(* IEC 61131-3 sources: io/test/Input, 8 files *)

(* ---- BinSignalExtTest.st ---- *)
USING AxUnit;
USING Simatic.Ax.IO.Input;
USING System.Timer;

NAMESPACE Simatic.Ax.IO.Input.Test

    /// Test fixture for BinSignalExt class
    /// Verifies extended binary signal functionality including:
    /// - All BinSignal features (signal reading, edge detection, inversion, quality status)
    /// - On-delay and off-delay timing functionality
    /// - Time-based signal filtering
    {TestFixture}
    CLASS BinSignalExtTest
        VAR
            o : BinSignalExt;  // Test object for BinSignalExt
            oStateLess : BinSignalExt;  // Stateless test object
        END_VAR

        /// Setup method called before each test
        /// Initializes test objects to ensure clean state
        {TestSetup}
        METHOD PUBLIC MyTestSetup
            o := oStateLess;
        END_METHOD

        /// Test basic signal reading - expects TRUE output when TRUE signal is read
        {Test}
        METHOD PUBLIC TestQ_And_expect_true
            o.ReadCyclic(signal := TRUE);
            Assert.Equal(expected := TRUE, actual := o.Q());
        END_METHOD

        {Test(isignal := FALSE, ienable := FALSE, idefault := FALSE, iexpq := FALSE, iexpqbad := TRUE)}
        {Test(isignal := FALSE, ienable := FALSE, idefault := TRUE, iexpq := TRUE, iexpqbad := TRUE)}
        {Test(isignal := FALSE, ienable := TRUE, idefault := FALSE, iexpq := FALSE, iexpqbad := FALSE)}
        {Test(isignal := FALSE, ienable := TRUE, idefault := TRUE, iexpq := FALSE, iexpqbad := FALSE)}

        {Test(isignal := TRUE, ienable := FALSE, idefault := FALSE, iexpq := FALSE, iexpqbad := TRUE)}
        {Test(isignal := TRUE, ienable := FALSE, idefault := TRUE, iexpq := TRUE, iexpqbad := TRUE)}
        {Test(isignal := TRUE, ienable := TRUE, idefault := FALSE, iexpq := TRUE, iexpqbad := FALSE)}
        {Test(isignal := TRUE, ienable := TRUE, idefault := TRUE, iexpq := TRUE, iexpqbad := FALSE)}

        METHOD PUBLIC  execute
            VAR_INPUT
                isignal : BOOL;
                ienable : BOOL;
                idefault : BOOL;
                iexpq : BOOL;
                iexpqbad : BOOL;
            END_VAR

            o.ReadCyclic(signal := iSignal, valid := iEnable, default := iDefault);
            AxUnit.Assert.Equal(expected := iExpQ, actual := o.Q());

        END_METHOD

        {Test(isignal := TRUE, ienable := TRUE, idefault := FALSE, iexpq := TRUE, iexpqris := TRUE, iexpqfal := FALSE, itestfallingedge := FALSE)}
        {Test(isignal := FALSE, ienable := TRUE, idefault := FALSE, iexpq := FALSE, iexpqris := FALSE, iexpqfal := TRUE, itestfallingedge := TRUE)}
        //-----------------------------------------------------------
        // test SetOff
        //-----------------------------------------------------------
        METHOD PUBLIC QRis2
            VAR_INPUT
                isignal : BOOL;
                ienable : BOOL;
                idefault : BOOL;
                iexpq : BOOL;
                iexpqris : BOOL;
                iexpqfal : BOOL;
                itestfallingedge : BOOL;
            END_VAR

            IF (iTestFallingEdge) then
                o.ReadCyclic(signal := TRUE, valid := iEnable, default := iDefault);
            END_IF;

            o.ReadCyclic(signal := iSignal, valid := iEnable, default := iDefault);
            AxUnit.Assert.Equal(expected := iExpQ, actual := o.Q());
            AxUnit.Assert.Equal(expected := iExpQRis, actual := o.QRis());
            AxUnit.Assert.Equal(expected := iExpQFal, actual := o.QFal());

            o.ReadCyclic(signal := iSignal, valid := iEnable, default := iDefault);
            AxUnit.Assert.Equal(expected := iExpQ, actual := o.Q());
            AxUnit.Assert.Equal(expected := FALSE, actual := o.QRis());
            AxUnit.Assert.Equal(expected := FALSE, actual := o.QFal());

        END_METHOD

        //-----------------------------------------------------------
        // test Q
        //-----------------------------------------------------------
        {Test}
        METHOD PUBLIC  Q
            VAR_TEMP
            END_VAR
            AxUnit.Assert.Equal(expected := FALSE, actual := o.Q());
            o.ReadCyclic(signal := TRUE);
            AxUnit.Assert.Equal(expected := TRUE, actual := o.Q());
            AxUnit.Assert.Equal(expected := FALSE, actual := o.QBad());
        END_METHOD

        //-----------------------------------------------------------
        // test QRis
        //-----------------------------------------------------------
        {Test}
        METHOD PUBLIC QRis
            AxUnit.Assert.Equal(expected := FALSE, actual := o.QRis());
            o.ReadCyclic(signal := TRUE);
            AxUnit.Assert.Equal(expected := TRUE, actual := o.QRis());
            o.ReadCyclic(signal := TRUE);
            AxUnit.Assert.Equal(expected := FALSE, actual := o.QRis());

            o.invert := TRUE;
            o.ReadCyclic(signal := TRUE);
            AxUnit.Assert.Equal(expected := FALSE, actual := o.QRis());
            o.ReadCyclic(signal := FALSE);
            AxUnit.Assert.Equal(expected := TRUE, actual := o.QRis());
            o.ReadCyclic(signal := TRUE);
            AxUnit.Assert.Equal(expected := FALSE, actual := o.QRis());

        END_METHOD
        //-----------------------------------------------------------
        // test QFal
        //-----------------------------------------------------------
        {Test}
        METHOD PUBLIC QFal

            o.ReadCyclic(signal := TRUE);
            AxUnit.Assert.Equal(expected := FALSE, actual := o.QFal());
            o.ReadCyclic(signal := FALSE);
            AxUnit.Assert.Equal(expected := TRUE, actual := o.QFal());
            o.ReadCyclic(signal := FALSE);
            AxUnit.Assert.Equal(expected := FALSE, actual := o.QFal());

            o.invert := TRUE;
            o.ReadCyclic(signal := FALSE);
            AxUnit.Assert.Equal(expected := FALSE, actual := o.QFal());
            o.ReadCyclic(signal := TRUE);
            AxUnit.Assert.Equal(expected := TRUE, actual := o.QFal());
            o.ReadCyclic(signal := FALSE);
            AxUnit.Assert.Equal(expected := FALSE, actual := o.QFal());

        END_METHOD

        //-----------------------------------------------------------
        // test QBad
        //-----------------------------------------------------------
        {Test}
        METHOD PUBLIC QBad

            o.ReadCyclic(signal := TRUE, valid := FALSE, default := FALSE);
            AxUnit.Assert.Equal(expected := TRUE, actual := o.QBad());
            AxUnit.Assert.Equal(expected := FALSE, actual := o.Q());

            o.ReadCyclic(signal := FALSE, valid := FALSE, default := TRUE);
            AxUnit.Assert.Equal(expected := TRUE, actual := o.QBad());
            AxUnit.Assert.Equal(expected := TRUE, actual := o.Q());

            o.invert  := TRUE;
            o.ReadCyclic(signal := TRUE, valid := FALSE, default := FALSE);
            AxUnit.Assert.Equal(expected := TRUE, actual := o.QBad());
            AxUnit.Assert.Equal(expected := FALSE, actual := o.Q());

            o.ReadCyclic(signal := FALSE, valid := FALSE, default := TRUE);
            AxUnit.Assert.Equal(expected := TRUE, actual := o.QBad());
            AxUnit.Assert.Equal(expected := TRUE, actual := o.Q());

            o.invert := TRUE;
            AxUnit.Assert.Equal(expected := TRUE, actual := o.IsInverted());
            o.ReadCyclic(signal := FALSE);
            AxUnit.Assert.Equal(expected := TRUE, actual := o.Q());

        END_METHOD

    END_CLASS
END_NAMESPACE

(* ---- BinSignalExtTest_TimeBehavior.st ---- *)
USING AxUnit;
USING Simatic.Ax.IO.Input;
USING System.Timer;
USING Simatic.Ax.Mocks;

NAMESPACE Simatic.Ax.IO.Input.Test

    /// Test fixture for timing behavior of BinSignalExt.
    /// Tests the correct handling of on-delay and off-delay logic in BinSignalExt.
    /// Input: None.
    /// Returns: None.
    {TestFixture}
    CLASS BinSignalExt_TimingTest
        VAR
            o, oStateLess : BinSignalExt;
        END_VAR

        /// Sets up the test environment for each test.
        /// Input: None.
        /// Returns: None.
        {TestSetup}
        METHOD PUBLIC TestSetup
            o := oStateLess;
        END_METHOD

        /// Verifies that Q() is FALSE immediately after signal becomes TRUE with on-delay active.
        /// Input: None.
        /// Returns: None.
        {Test}
        METHOD PUBLIC TestOnDelay_After_signal_true_expect_false
            AxUnit.Mocking.Mock(NAME_OF(OnDelay), NAME_OF(OnDelayMock_false));
            o.ondelay := T#10ms;
            o.ReadCyclic(signal := TRUE);
            Assert.Equal(expected := FALSE, actual := o.Q());
        END_METHOD

        /// Verifies that Q() is TRUE after signal is TRUE and on-delay has elapsed.
        /// Input: None.
        /// Returns: None.
        {Test}
        METHOD PUBLIC TestOnDelay_10ms_After_signal_true_expect_true
            AxUnit.Mocking.Mock(NAME_OF(OnDelay), NAME_OF(OnDelayMock_true));
            o.ondelay := T#10ms;
            o.ReadCyclic(signal := TRUE);
            Assert.Equal(expected := TRUE, actual := o.Q());
        END_METHOD

        /// Verifies that Q() is TRUE after on-delay, and becomes FALSE when signal goes to FALSE.
        /// Input: None.
        /// Returns: None.
        {Test}
        METHOD PUBLIC TestOnDelay_10ms_signal_goes_to_False_expect_false
            AxUnit.Mocking.Mock(NAME_OF(OnDelay), NAME_OF(OnDelayMock_true));
            o.ondelay := T#10ms;
            o.ReadCyclic(signal := TRUE);
            Assert.Equal(expected := TRUE, actual := o.Q());
            AxUnit.Mocking.Mock(NAME_OF(OnDelay), NAME_OF(OnDelayMock_false));
            o.ReadCyclic(signal := FALSE);
            Assert.Equal(expected := FALSE, actual := o.Q());
        END_METHOD

        /// Verifies that Q() remains TRUE after signal goes FALSE if off-delay is active, then becomes FALSE after off-delay.
        /// Input: None.
        /// Returns: None.
        {Test}
        METHOD PUBLIC TestOffDelay_10ms_After_signal_true_expect_true
            AxUnit.Mocking.Mock(NAME_OF(OffDelay), NAME_OF(OffDelayMock_true));
            o.offdelay := T#10ms;
            o.ReadCyclic(signal := TRUE);
            o.ReadCyclic(signal := FALSE);
            Assert.Equal(expected := TRUE, actual := o.Q());

            AxUnit.Mocking.Mock('System.Timer.OffDelay', 'Simatic.Ax.Mocks.OffDelayMock_false');
            o.ReadCyclic(signal := FALSE);
            Assert.Equal(expected := FALSE, actual := o.Q());
        END_METHOD
    END_CLASS
END_NAMESPACE

(* ---- BinSignalTest.st ---- *)
USING AxUnit;
USING Simatic.Ax.IO.Input;
USING System.Timer;

NAMESPACE Simatic.Ax.IO.Input.Test

    /// Test fixture for BinSignal class
    /// Verifies binary signal input functionality including:
    /// - Signal reading and state management
    /// - Edge detection (rising and falling edges)
    /// - Signal inversion
    /// - Quality status (QBad) handling
    /// - Change detection
    {TestFixture}
    CLASS BinSignalTest
        VAR
            o : BinSignal;   // Test object for BinSignal
            oStateLess : BinSignalExt;  // Stateless test object
        END_VAR

        /// Setup method called before each test
        /// Initializes test objects to ensure clean state
        {TestSetup}
        METHOD PUBLIC MyTestSetup
            o := oStateLess;
        END_METHOD

        /// Test basic signal reading - expects TRUE output when TRUE signal is read
        {Test}
        METHOD PUBLIC TestQ_And_expect_true
            o.ReadCyclic(signal := TRUE);
            Assert.Equal(expected := TRUE, actual := o.Q());
        END_METHOD

        /// Parameterized test for signal reading with different valid/invalid combinations
        /// Tests all combinations of signal value, validity flag, and default value
        /// Verifies that Q() returns correct value and QBad() reflects validity status
        {Test(isignal := FALSE, ienable := FALSE, idefault := FALSE, iexpq := FALSE, iexpqbad := TRUE)}
        {Test(isignal := FALSE, ienable := FALSE, idefault := TRUE, iexpq := TRUE, iexpqbad := TRUE)}
        {Test(isignal := FALSE, ienable := TRUE, idefault := FALSE, iexpq := FALSE, iexpqbad := FALSE)}
        {Test(isignal := FALSE, ienable := TRUE, idefault := TRUE, iexpq := FALSE, iexpqbad := FALSE)}

        {Test(isignal := TRUE, ienable := FALSE, idefault := FALSE, iexpq := FALSE, iexpqbad := TRUE)}
        {Test(isignal := TRUE, ienable := FALSE, idefault := TRUE, iexpq := TRUE, iexpqbad := TRUE)}
        {Test(isignal := TRUE, ienable := TRUE, idefault := FALSE, iexpq := TRUE, iexpqbad := FALSE)}
        {Test(isignal := TRUE, ienable := TRUE, idefault := TRUE, iexpq := TRUE, iexpqbad := FALSE)}

        METHOD PUBLIC execute
            VAR_INPUT
                isignal : BOOL;
                ienable : BOOL;
                idefault : BOOL;
                iexpq : BOOL;
                iexpqbad : BOOL;
            END_VAR

            o.ReadCyclic(signal := iSignal, valid := iEnable, default := iDefault);
            AxUnit.Assert.Equal(expected := iExpQ, actual := o.Q());

        END_METHOD

        /// Parameterized test for edge detection (rising and falling edges)
        /// Verifies QRis() and QFal() correctly detect signal transitions
        {Test(isignal := TRUE, ienable := TRUE, idefault := FALSE, iexpq := TRUE, iexpqris := TRUE, iexpqfal := FALSE, itestfallingedge := FALSE)}
        {Test(isignal := FALSE, ienable := TRUE, idefault := FALSE, iexpq := FALSE, iexpqris := FALSE, iexpqfal := TRUE, itestfallingedge := TRUE)}
        METHOD PUBLIC QRis2
            VAR_INPUT
                isignal : BOOL;
                ienable : BOOL;
                idefault : BOOL;
                iexpq : BOOL;
                iexpqris : BOOL;
                iexpqfal : BOOL;
                itestfallingedge : BOOL;
            END_VAR

            IF (iTestFallingEdge) then
                o.ReadCyclic(signal := TRUE, valid := iEnable, default := iDefault);
            END_IF;

            o.ReadCyclic(signal := iSignal, valid := iEnable, default := iDefault);
            AxUnit.Assert.Equal(expected := iExpQ, actual := o.Q());
            AxUnit.Assert.Equal(expected := iExpQRis, actual := o.QRis());
            AxUnit.Assert.Equal(expected := iExpQFal, actual := o.QFal());

            o.ReadCyclic(signal := iSignal, valid := iEnable, default := iDefault);
            AxUnit.Assert.Equal(expected := iExpQ, actual := o.Q());
            AxUnit.Assert.Equal(expected := FALSE, actual := o.QRis());
            AxUnit.Assert.Equal(expected := FALSE, actual := o.QFal());

        END_METHOD

        /// Test Q() method - verifies signal state reading and QBad status
        {Test}
        METHOD PUBLIC Q
            VAR_TEMP
            END_VAR
            AxUnit.Assert.Equal(expected := FALSE, actual := o.Q());
            o.ReadCyclic(signal := TRUE);
            AxUnit.Assert.Equal(expected := TRUE, actual := o.Q());
            AxUnit.Assert.Equal(expected := FALSE, actual := o.QBad());
        END_METHOD

        /// Test QRis() method - verifies rising edge detection with and without inversion
        {Test}
        METHOD PUBLIC QRis
            AxUnit.Assert.Equal(expected := FALSE, actual := o.QRis());
            o.ReadCyclic(signal := TRUE);
            AxUnit.Assert.Equal(expected := TRUE, actual := o.QRis());
            o.ReadCyclic(signal := TRUE);
            AxUnit.Assert.Equal(expected := FALSE, actual := o.QRis());

            o.invert := TRUE;
            o.ReadCyclic(signal := TRUE);
            AxUnit.Assert.Equal(expected := FALSE, actual := o.QRis());
            o.ReadCyclic(signal := FALSE);
            AxUnit.Assert.Equal(expected := TRUE, actual := o.QRis());
            o.ReadCyclic(signal := TRUE);
            AxUnit.Assert.Equal(expected := FALSE, actual := o.QRis());

        END_METHOD
        /// Test QFal() method - verifies falling edge detection with and without inversion
        {Test}
        METHOD PUBLIC QFal

            o.ReadCyclic(signal := TRUE);
            AxUnit.Assert.Equal(expected := FALSE, actual := o.QFal());
            o.ReadCyclic(signal := FALSE);
            AxUnit.Assert.Equal(expected := TRUE, actual := o.QFal());
            o.ReadCyclic(signal := FALSE);
            AxUnit.Assert.Equal(expected := FALSE, actual := o.QFal());

            o.invert := TRUE;
            o.ReadCyclic(signal := FALSE);
            AxUnit.Assert.Equal(expected := FALSE, actual := o.QFal());
            o.ReadCyclic(signal := TRUE);
            AxUnit.Assert.Equal(expected := TRUE, actual := o.QFal());
            o.ReadCyclic(signal := FALSE);
            AxUnit.Assert.Equal(expected := FALSE, actual := o.QFal());

        END_METHOD

        /// Test QBad() method - verifies quality status handling with valid/invalid signals
        /// Tests default value behavior and signal inversion with quality status
        {Test}
        METHOD PUBLIC QBad

            o.ReadCyclic(signal := TRUE, valid := FALSE, default := FALSE);
            AxUnit.Assert.Equal(expected := TRUE, actual := o.QBad());
            AxUnit.Assert.Equal(expected := FALSE, actual := o.Q());

            o.ReadCyclic(signal := FALSE, valid := FALSE, default := TRUE);
            AxUnit.Assert.Equal(expected := TRUE, actual := o.QBad());
            AxUnit.Assert.Equal(expected := TRUE, actual := o.Q());

            o.invert  := TRUE;
            o.ReadCyclic(signal := TRUE, valid := FALSE, default := FALSE);
            AxUnit.Assert.Equal(expected := TRUE, actual := o.QBad());
            AxUnit.Assert.Equal(expected := FALSE, actual := o.Q());

            o.ReadCyclic(signal := FALSE, valid := FALSE, default := TRUE);
            AxUnit.Assert.Equal(expected := TRUE, actual := o.QBad());
            AxUnit.Assert.Equal(expected := TRUE, actual := o.Q());

            o.invert := TRUE;
            AxUnit.Assert.Equal(expected := TRUE, actual := o.IsInverted());
            o.ReadCyclic(signal := FALSE);
            AxUnit.Assert.Equal(expected := TRUE, actual := o.Q());

        END_METHOD

        /// Test HasChanged() method - verifies change detection between consecutive reads
        {Test}
        METHOD PUBLIC HasChanged

            o.ReadCyclic(signal := TRUE, valid := TRUE, default := FALSE);
            o.ReadCyclic(signal := TRUE, valid := TRUE, default := FALSE);
            AxUnit.Assert.Equal(expected := FALSE, actual := o.HasChanged());

            o.ReadCyclic(signal := FALSE, valid := TRUE, default := FALSE);
            o.ReadCyclic(signal := FALSE, valid := TRUE, default := FALSE);
            AxUnit.Assert.Equal(expected := FALSE, actual := o.HasChanged());

            o.ReadCyclic(signal := FALSE, valid := TRUE, default := FALSE);
            o.ReadCyclic(signal := TRUE, valid := TRUE, default := FALSE);
            AxUnit.Assert.Equal(expected := TRUE, actual := o.HasChanged());

            o.ReadCyclic(signal := TRUE, valid := TRUE, default := FALSE);
            o.ReadCyclic(signal := FALSE, valid := TRUE, default := FALSE);
            AxUnit.Assert.Equal(expected := TRUE, actual := o.HasChanged());

        END_METHOD

    END_CLASS
END_NAMESPACE

(* ---- DintInputTest.st ---- *)
USING Simatic.Ax.IO.Input;
USING AxUnit;

NAMESPACE Simatic.Ax.IO.Input.Test

    /// Test fixture for DintInput class
    /// Verifies double integer (DINT) input functionality including:
    /// - Signal reading with valid/invalid status
    /// - Default value handling when signal is invalid
    /// - QBad status management
    /// - Change detection with and without tolerance
    /// - MIN/MAX constant values
    {TestFixture}
    CLASS DintInputTest
        VAR
            o : DintInput;  // Test object for DintInput
            oMinMaxTest : DintInput;  // Test object for MIN/MAX verification
        END_VAR

        /// Parameterized test for different signal values and validity combinations
        /// Verifies Q() returns correct value based on validity and QBad() reflects status
        {Test(signalValue := DINT#0, isValid := FALSE, defaultValue := DINT#0, expectedValueWhenQBad := DINT#0, expectedQBad := TRUE)}
        {Test(signalValue := DINT#0, isValid := FALSE, defaultValue := DINT#1, expectedValueWhenQBad := DINT#1, expectedQBad := TRUE)}
        {Test(signalValue := DINT#0, isValid := TRUE, defaultValue := DINT#0, expectedValueWhenQBad := DINT#0, expectedQBad := FALSE)}
        {Test(signalValue := DINT#0, isValid := TRUE, defaultValue := DINT#1, expectedValueWhenQBad := DINT#0, expectedQBad := FALSE)}

        {Test(signalValue := DINT#100, isValid := FALSE, defaultValue := DINT#0, expectedValueWhenQBad := DINT#0, expectedQBad := TRUE)}
        {Test(signalValue := DINT#100, isValid := FALSE, defaultValue := DINT#1, expectedValueWhenQBad := DINT#1, expectedQBad := TRUE)}
        {Test(signalValue := DINT#100, isValid := TRUE, defaultValue := DINT#0, expectedValueWhenQBad := DINT#100, expectedQBad := FALSE)}
        {Test(signalValue := DINT#100, isValid := TRUE, defaultValue := DINT#1, expectedValueWhenQBad := DINT#100, expectedQBad := FALSE)}
        METHOD PUBLIC Check_different_values_and_results
            VAR_INPUT
                signalValue : DINT;
                isValid : BOOL;
                defaultValue : DINT;
                expectedValueWhenQBad : DINT;
                expectedQBad : BOOL;
            END_VAR

            o.ReadCyclic(value := signalValue, valid := isValid, default := defaultValue);
            Assert.Equal(expected := expectedValueWhenQBad, actual := o.Q());
            Assert.Equal(expected := expectedQBad, actual := o.QBad());
        END_METHOD

        /// Test MIN and MAX constants for DINT data type
        {Test}
        METHOD PUBLIC CheckMinMax
            Assert.Equal(expected := DINT#-2147483648, actual := oMinMaxTest.Min);
            Assert.Equal(expected := DINT#2147483647, actual := oMinMaxTest.Max);
        END_METHOD

        /// Test change detection without tolerance
        /// Verifies HasChanged() detects any value change
        {Test(signalValue := DINT#100, newSignalValue := DINT#100, expectedHasChanged := FALSE)}
        {Test(signalValue := DINT#100, newSignalValue := DINT#101, expectedHasChanged := TRUE)}
        METHOD PUBLIC CheckHasChanged
            VAR_INPUT
                signalValue : DINT;
                newSignalValue : DINT;
                expectedHasChanged : BOOL;
            END_VAR

            o.ReadCyclic(value := signalValue, valid := TRUE, default := 0);
            o.ReadCyclic(value := newSignalValue, valid := TRUE, default := 0);
            Assert.Equal(expected := expectedHasChanged, actual := o.HasChanged());
        END_METHOD

        /// Test change detection with tolerance
        /// Verifies HasChanged() only triggers when change exceeds tolerance
        {Test(signalValue := DINT#100, newSignalValue := DINT#100, tolerance := DINT#10, expectedHasChanged := FALSE)}
        {Test(signalValue := DINT#100, newSignalValue := DINT#111, tolerance := DINT#10, expectedHasChanged := TRUE)}
        METHOD PUBLIC CheckHasChangedWithTolerance
            VAR_INPUT
                signalValue : DINT;
                newSignalValue : DINT;
                tolerance : DINT;
                expectedHasChanged : BOOL;
            END_VAR

            o.ReadCyclic(value := signalValue, valid := TRUE, default := 0);
            o.ReadCyclic(value := newSignalValue, valid := TRUE, default := 0, tolerance := tolerance);
            Assert.Equal(expected := expectedHasChanged, actual := o.HasChanged());
        END_METHOD
    END_CLASS
END_NAMESPACE

(* ---- IntInputTest.st ---- *)
USING Simatic.Ax.IO.Input;
USING AxUnit;

NAMESPACE Simatic.Ax.IO.Input.Test

    /// Test fixture for IntInput class
    /// Verifies integer (INT) input functionality including:
    /// - Signal reading with valid/invalid status
    /// - Default value handling when signal is invalid
    /// - QBad status management
    /// - Change detection with and without tolerance
    /// - MIN/MAX constant values
    {TestFixture}
    CLASS IntInputTest
        VAR
            o : IntInput;  // Test object for IntInput
            oMinMaxTest : IntInput;  // Test object for MIN/MAX verification
        END_VAR

        /// Parameterized test for different signal values and validity combinations
        /// Verifies Q() returns correct value based on validity and QBad() reflects status
        {Test(signalValue := INT#0, isValid := FALSE, defaultValue := INT#0, expectedValueWhenQBad := INT#0, expectedQBad := TRUE)}
        {Test(signalValue := INT#0, isValid := FALSE, defaultValue := INT#1, expectedValueWhenQBad := INT#1, expectedQBad := TRUE)}
        {Test(signalValue := INT#0, isValid := TRUE, defaultValue := INT#0, expectedValueWhenQBad := INT#0, expectedQBad := FALSE)}
        {Test(signalValue := INT#0, isValid := TRUE, defaultValue := INT#1, expectedValueWhenQBad := INT#0, expectedQBad := FALSE)}

        {Test(signalValue := INT#100, isValid := FALSE, defaultValue := INT#0, expectedValueWhenQBad := INT#0, expectedQBad := TRUE)}
        {Test(signalValue := INT#100, isValid := FALSE, defaultValue := INT#1, expectedValueWhenQBad := INT#1, expectedQBad := TRUE)}
        {Test(signalValue := INT#100, isValid := TRUE, defaultValue := INT#0, expectedValueWhenQBad := INT#100, expectedQBad := FALSE)}
        {Test(signalValue := INT#100, isValid := TRUE, defaultValue := INT#1, expectedValueWhenQBad := INT#100, expectedQBad := FALSE)}
        METHOD PUBLIC Check_different_values_and_results
            VAR_INPUT
                signalValue : INT;
                isValid : BOOL;
                defaultValue : INT;
                expectedValueWhenQBad : INT;
                expectedQBad : BOOL;
            END_VAR

            o.ReadCyclic(value := signalValue, valid := isValid, default := defaultValue);
            Assert.Equal(expected := expectedValueWhenQBad, actual := o.Q());
            Assert.Equal(expected := expectedQBad, actual := o.QBad());
        END_METHOD

        /// Test MIN and MAX constants for INT data type
        {Test}
        METHOD PUBLIC CheckMinMax
            AxUnit.Assert.Equal(expected := -32768, actual := oMinMaxTest.Min);
            AxUnit.Assert.Equal(expected :=  32767, actual := oMinMaxTest.Max);

        END_METHOD

        /// Test change detection without tolerance
        /// Verifies HasChanged() detects any value change
        {Test(signalValue := INT#100, newSignalValue := INT#100, expectedHasChanged := FALSE)}
        {Test(signalValue := INT#100, newSignalValue := INT#101, expectedHasChanged := TRUE)}
        METHOD PUBLIC CheckHasChanged
            VAR_INPUT
                signalValue : INT;
                newSignalValue : INT;
                expectedHasChanged : BOOL;
            END_VAR

            o.ReadCyclic(value := signalValue, valid := TRUE, default := 0);
            o.ReadCyclic(value := newSignalValue, valid := TRUE, default := 0);
            Assert.Equal(expected := expectedHasChanged, actual := o.HasChanged());
        END_METHOD

        /// Test change detection with tolerance
        /// Verifies HasChanged() only triggers when change exceeds tolerance
        {Test(signalValue := INT#100, newSignalValue := INT#100, tolerance := 10, expectedHasChanged := FALSE)}
        {Test(signalValue := INT#100, newSignalValue := INT#111, tolerance := 10, expectedHasChanged := TRUE)}
        METHOD PUBLIC CheckHasChangedWithTolerance
            VAR_INPUT
                signalValue : INT;
                newSignalValue : INT;
                tolerance : INT;
                expectedHasChanged : BOOL;
            END_VAR

            o.ReadCyclic(value := signalValue, valid := TRUE, default := 0);
            o.ReadCyclic(value := newSignalValue, valid := TRUE, default := 0, tolerance := tolerance);
            Assert.Equal(expected := expectedHasChanged, actual := o.HasChanged());
        END_METHOD
    END_CLASS
END_NAMESPACE

(* ---- LRealInputTest.st ---- *)
USING Simatic.Ax.IO.Input;
USING AxUnit;

NAMESPACE Simatic.Ax.IO.Input.Test

    /// Test fixture for LRealInput class
    /// Verifies long real (LREAL) double precision floating-point input functionality including:
    /// - Signal reading with valid/invalid status (from LWORD hardware format and LREAL software format)
    /// - Default value handling when signal is invalid
    /// - QBad status management
    /// - Change detection with tolerance for floating-point values
    /// - MIN/MAX constant values
    {TestFixture}
    CLASS LRealInputTest
        VAR
            o : LRealInput;  // Test object for LRealInput
            oMinMaxTest : LRealInput;  // Test object for MIN/MAX verification
        END_VAR

        /// Parameterized test for different signal values and validity combinations
        /// Tests reading from LWORD hardware format (TO_LWORD conversion)
        /// Verifies Q() returns correct value based on validity and QBad() reflects status
        {Test(signalValue := LREAL#0.0, isValid := FALSE, defaultValue := LREAL#0.0, expectedValueWhenQBad := LREAL#0.0, expectedQBad := TRUE)}
        {Test(signalValue := LREAL#0.0, isValid := FALSE, defaultValue := LREAL#1.0, expectedValueWhenQBad := LREAL#1.0, expectedQBad := TRUE)}
        {Test(signalValue := LREAL#0.0, isValid := TRUE, defaultValue := LREAL#0.0, expectedValueWhenQBad := LREAL#0.0, expectedQBad := FALSE)}
        {Test(signalValue := LREAL#0.0, isValid := TRUE, defaultValue := LREAL#1.0, expectedValueWhenQBad := LREAL#0.0, expectedQBad := FALSE)}

        {Test(signalValue := LREAL#100.0, isValid := FALSE, defaultValue := LREAL#0.0, expectedValueWhenQBad := LREAL#0.0, expectedQBad := TRUE)}
        {Test(signalValue := LREAL#100.0, isValid := FALSE, defaultValue := LREAL#1.0, expectedValueWhenQBad := LREAL#1.0, expectedQBad := TRUE)}
        {Test(signalValue := LREAL#100.0, isValid := TRUE, defaultValue := LREAL#0.0, expectedValueWhenQBad := LREAL#100.0, expectedQBad := FALSE)}
        {Test(signalValue := LREAL#100.0, isValid := TRUE, defaultValue := LREAL#1.0, expectedValueWhenQBad := LREAL#100.0, expectedQBad := FALSE)}
        METHOD PUBLIC Check_different_values_and_results
            VAR_INPUT
                signalValue : LREAL;
                isValid : BOOL;
                defaultValue : LREAL;
                expectedValueWhenQBad : LREAL;
                expectedQBad : BOOL;
            END_VAR

            o.ReadCyclic(value := TO_LWORD(signalValue), valid := isValid, default := defaultValue);
            Assert.Equal(expected := expectedValueWhenQBad, actual := o.Q());
            Assert.Equal(expected := expectedQBad, actual := o.QBad());
        END_METHOD

        /// Parameterized test for LREAL software format input
        /// Tests reading directly from LREAL values (software sources)
        /// Verifies Q() returns correct value based on validity and QBad() reflects status
        {Test(signalValue := LREAL#0.0, isValid := FALSE, defaultValue := LREAL#0.0, expectedValueWhenQBad := LREAL#0.0, expectedQBad := TRUE)}
        {Test(signalValue := LREAL#0.0, isValid := FALSE, defaultValue := LREAL#1.0, expectedValueWhenQBad := LREAL#1.0, expectedQBad := TRUE)}
        {Test(signalValue := LREAL#0.0, isValid := TRUE, defaultValue := LREAL#0.0, expectedValueWhenQBad := LREAL#0.0, expectedQBad := FALSE)}
        {Test(signalValue := LREAL#0.0, isValid := TRUE, defaultValue := LREAL#1.0, expectedValueWhenQBad := LREAL#0.0, expectedQBad := FALSE)}

        {Test(signalValue := LREAL#100.0, isValid := FALSE, defaultValue := LREAL#0.0, expectedValueWhenQBad := LREAL#0.0, expectedQBad := TRUE)}
        {Test(signalValue := LREAL#100.0, isValid := FALSE, defaultValue := LREAL#1.0, expectedValueWhenQBad := LREAL#1.0, expectedQBad := TRUE)}
        {Test(signalValue := LREAL#100.0, isValid := TRUE, defaultValue := LREAL#0.0, expectedValueWhenQBad := LREAL#100.0, expectedQBad := FALSE)}
        {Test(signalValue := LREAL#100.0, isValid := TRUE, defaultValue := LREAL#1.0, expectedValueWhenQBad := LREAL#100.0, expectedQBad := FALSE)}
        METHOD PUBLIC Check_different_LREAL_values_and_results
            VAR_INPUT
                signalValue : LREAL;
                isValid : BOOL;
                defaultValue : LREAL;
                expectedValueWhenQBad : LREAL;
                expectedQBad : BOOL;
            END_VAR

            o.ReadCyclic(value := signalValue, valid := isValid, default := defaultValue);
            Assert.Equal(expected := expectedValueWhenQBad, actual := o.Q());
            Assert.Equal(expected := expectedQBad, actual := o.QBad());
        END_METHOD

        /// Test MIN and MAX constants for LREAL data type
        {Test}
        METHOD PUBLIC CheckMinMax
            Assert.Equal(expected := LREAL#1.79769313486231e+308, actual := oMinMaxTest.Max);
            Assert.Equal(expected :=  LREAL#-1.79769313486231e+308, actual := oMinMaxTest.Min);
        END_METHOD

        /// Test change detection with tolerance for double precision floating-point values
        /// Verifies HasChanged() only triggers when change exceeds tolerance
        /// Important for filtering minor floating-point fluctuations
        {Test(signalValue := LREAL#100.0, newSignalValue := LREAL#100.0, tolerance := 0.1, expectedHasChanged := FALSE)}
        {Test(signalValue := LREAL#100.0, newSignalValue := LREAL#101.0, tolerance := 0.1, expectedHasChanged := TRUE)}
        {Test(signalValue := LREAL#100.0, newSignalValue := LREAL#100.2, tolerance := 0.1, expectedHasChanged := TRUE)}
        {Test(signalValue := LREAL#100.0, newSignalValue := LREAL#100.05, tolerance := 0.1, expectedHasChanged := FALSE)}
        METHOD PUBLIC CheckHasChanged
            VAR_INPUT
                signalValue : LREAL;
                newSignalValue : LREAL;
                tolerance : LREAL;
                expectedHasChanged : BOOL;
            END_VAR

            o.ReadCyclic(value := signalValue, valid := TRUE, default := 0);
            o.ReadCyclic(value := newSignalValue, valid := TRUE, default := 0, tolerance := tolerance);
            Assert.Equal(expected := expectedHasChanged, actual := o.HasChanged());
        END_METHOD
    END_CLASS
END_NAMESPACE

(* ---- RealInputTest.st ---- *)
USING Simatic.Ax.IO.Input;
USING AxUnit;

NAMESPACE Simatic.Ax.IO.Input.Test

    /// Test fixture for RealInput class
    /// Verifies real (REAL) floating-point input functionality including:
    /// - Signal reading with valid/invalid status (from DWORD hardware format)
    /// - Default value handling when signal is invalid
    /// - QBad status management
    /// - Change detection with tolerance for floating-point values
    /// - MIN/MAX constant values
    {TestFixture}
    CLASS RealInputTest
        VAR
            o : RealInput;  // Test object for RealInput
            oMinMaxTest : RealInput;  // Test object for MIN/MAX verification
        END_VAR

        /// Parameterized test for different signal values and validity combinations
        /// Tests reading from DWORD hardware format (TO_DWORD conversion)
        /// Verifies Q() returns correct value based on validity and QBad() reflects status
        {Test(signalValue := REAL#0.0, isValid := FALSE, defaultValue := REAL#0.0, expectedValueWhenQBad := REAL#0.0, expectedQBad := TRUE)}
        {Test(signalValue := REAL#0.0, isValid := FALSE, defaultValue := REAL#1.0, expectedValueWhenQBad := REAL#1.0, expectedQBad := TRUE)}
        {Test(signalValue := REAL#0.0, isValid := TRUE, defaultValue := REAL#0.0, expectedValueWhenQBad := REAL#0.0, expectedQBad := FALSE)}
        {Test(signalValue := REAL#0.0, isValid := TRUE, defaultValue := REAL#1.0, expectedValueWhenQBad := REAL#0.0, expectedQBad := FALSE)}

        {Test(signalValue := REAL#100.0, isValid := FALSE, defaultValue := REAL#0.0, expectedValueWhenQBad := REAL#0.0, expectedQBad := TRUE)}
        {Test(signalValue := REAL#100.0, isValid := FALSE, defaultValue := REAL#1.0, expectedValueWhenQBad := REAL#1.0, expectedQBad := TRUE)}
        {Test(signalValue := REAL#100.0, isValid := TRUE, defaultValue := REAL#0.0, expectedValueWhenQBad := REAL#100.0, expectedQBad := FALSE)}
        {Test(signalValue := REAL#100.0, isValid := TRUE, defaultValue := REAL#1.0, expectedValueWhenQBad := REAL#100.0, expectedQBad := FALSE)}
        METHOD PUBLIC Check_different_values_and_results
            VAR_INPUT
                signalValue : REAL;
                isValid : BOOL;
                defaultValue : REAL;
                expectedValueWhenQBad : REAL;
                expectedQBad : BOOL;
            END_VAR

            o.ReadCyclic(value := TO_DWORD(signalValue), valid := isValid, default := defaultValue);
            Assert.Equal(expected := expectedValueWhenQBad, actual := o.Q());
            Assert.Equal(expected := expectedQBad, actual := o.QBad());
        END_METHOD

        /// Test MIN and MAX constants for REAL data type
        {Test}
        METHOD PUBLIC CheckMinMax
            Assert.Equal(expected := REAL#+3.402823e+38, actual := oMinMaxTest.Max);
            Assert.Equal(expected :=  REAL#-3.402823e+38, actual := oMinMaxTest.Min);
        END_METHOD

        /// Test change detection with tolerance for floating-point values
        /// Verifies HasChanged() only triggers when change exceeds tolerance
        /// Important for filtering minor floating-point fluctuations
        {Test(signalValue := REAL#100.0, newSignalValue := REAL#100.0, tolerance := REAL#0.1, expectedHasChanged := FALSE)}
        {Test(signalValue := REAL#100.0, newSignalValue := REAL#101.0, tolerance := REAL#0.1, expectedHasChanged := TRUE)}
        {Test(signalValue := REAL#100.0, newSignalValue := REAL#100.2, tolerance := REAL#0.1, expectedHasChanged := TRUE)}
        {Test(signalValue := REAL#100.0, newSignalValue := REAL#100.05, tolerance := REAL#0.1, expectedHasChanged := FALSE)}
        METHOD PUBLIC CheckHasChanged
            VAR_INPUT
                signalValue : REAL;
                newSignalValue : REAL;
                tolerance : REAL;
                expectedHasChanged : BOOL;
            END_VAR

            o.ReadCyclic(value := signalValue, valid := TRUE, default := 0);
            o.ReadCyclic(value := newSignalValue, valid := TRUE, default := 0, tolerance := tolerance);
            Assert.Equal(expected := expectedHasChanged, actual := o.HasChanged());
        END_METHOD
    END_CLASS
END_NAMESPACE

(* ---- WordInputTest.st ---- *)
USING Simatic.Ax.IO.Input;
USING AxUnit;

NAMESPACE Simatic.Ax.IO.Input.Test

    /// Test fixture for WordInput class
    /// Verifies word (WORD) input functionality including:
    /// - Signal reading with valid/invalid status
    /// - Default value handling when signal is invalid
    /// - QBad status management
    /// - Change detection (any bit change triggers)
    /// - MIN/MAX constant values
    {TestFixture}
    CLASS WordInputTest
        VAR
            o : WordInput;  // Test object for WordInput
            oMinMaxTest : WordInput;  // Test object for MIN/MAX verification
        END_VAR

        /// Parameterized test for different signal values and validity combinations
        /// Verifies Q() returns correct value based on validity and QBad() reflects status
        {Test(signalValue := WORD#16#0, isValid := FALSE, defaultValue := WORD#16#0, expectedValueWhenQBad := WORD#16#0, expectedQBad := TRUE)}
        {Test(signalValue := WORD#16#0, isValid := FALSE, defaultValue := WORD#16#1, expectedValueWhenQBad := WORD#16#1, expectedQBad := TRUE)}
        {Test(signalValue := WORD#16#0, isValid := TRUE, defaultValue := WORD#16#0, expectedValueWhenQBad := WORD#16#0, expectedQBad := FALSE)}
        {Test(signalValue := WORD#16#0, isValid := TRUE, defaultValue := WORD#16#1, expectedValueWhenQBad := WORD#16#0, expectedQBad := FALSE)}

        {Test(signalValue := WORD#16#100, isValid := FALSE, defaultValue := WORD#16#0, expectedValueWhenQBad := WORD#16#0, expectedQBad := TRUE)}
        {Test(signalValue := WORD#16#100, isValid := FALSE, defaultValue := WORD#16#1, expectedValueWhenQBad := WORD#16#1, expectedQBad := TRUE)}
        {Test(signalValue := WORD#16#100, isValid := TRUE, defaultValue := WORD#16#0, expectedValueWhenQBad := WORD#16#100, expectedQBad := FALSE)}
        {Test(signalValue := WORD#16#100, isValid := TRUE, defaultValue := WORD#16#1, expectedValueWhenQBad := WORD#16#100, expectedQBad := FALSE)}
        METHOD PUBLIC Check_different_values_and_results
            VAR_INPUT
                signalValue : WORD;
                isValid : BOOL;
                defaultValue : WORD;
                expectedValueWhenQBad : WORD;
                expectedQBad : BOOL;
            END_VAR

            o.ReadCyclic(value := signalValue, valid := isValid, default := defaultValue);
            Assert.Equal(expected := expectedValueWhenQBad, actual := o.Q());
            Assert.Equal(expected := expectedQBad, actual := o.QBad());
        END_METHOD

        /// Test MIN and MAX constants for WORD data type
        {Test}
        METHOD PUBLIC CheckMinMax
            AxUnit.Assert.Equal(expected := WORD#16#0, actual := oMinMaxTest.Min);
            AxUnit.Assert.Equal(expected := WORD#16#FFFF, actual := oMinMaxTest.Max);

        END_METHOD

        /// Test change detection - triggers on any bit change
        /// Verifies HasChanged() detects any value change
        {Test(signalValue := WORD#100, newSignalValue := WORD#100, expectedHasChanged := FALSE)}
        {Test(signalValue := WORD#100, newSignalValue := WORD#101, expectedHasChanged := TRUE)}
        METHOD PUBLIC CheckHasChanged
            VAR_INPUT
                signalValue : WORD;
                newSignalValue : WORD;
                expectedHasChanged : BOOL;
            END_VAR

            o.ReadCyclic(value := signalValue, valid := TRUE, default := WORD#16#0);
            o.ReadCyclic(value := newSignalValue, valid := TRUE, default := WORD#16#0);
            Assert.Equal(expected := expectedHasChanged, actual := o.HasChanged());
        END_METHOD
    END_CLASS
END_NAMESPACE
